{attribute 'linkalways'} 
{attribute 'no_explicit_call' := 'This FB is a CLASS and must be accessed using methods or properties'}
{attribute 'enable_dynamic_creation'}
FUNCTION_BLOCK Node_F_VN_GetAt_UDINT EXTENDS VisionNode
VAR
    ipContainer : _ITcVnContainer;
    nElement : _UDINT(0);
    nIndex : _ULINT(0);
    hrPrev : _HRESULT(S_OK);
    hresult : _HRESULT(S_OK);
END_VAR

METHOD PUBLIC  Clone : I_Node
VAR
	pNode : POINTER TO Node_F_VN_GetAt_UDINT;
END_VAR
pNode := __NEW(Node_F_VN_GetAt_UDINT);
Clone := pNode^;
END_METHOD

METHOD FB_init : BOOL
VAR_INPUT
	bInitRetains : BOOL; // if TRUE, the retain variables are initialized (warm start / cold start)
	bInCopyCode : BOOL;  // if TRUE, the instance afterwards gets moved into the copy code (online change)
END_VAR
AddInput('ipContainer', ipContainer);
AddInput('nIndex', nIndex);
AddInput('hrPrev', hrPrev);
AddOutput('nElement', nElement);
AddOutput('hresult',hresult);
END_METHOD

METHOD PROTECTED OnExecute : HRESULT
hresult.Value := F_VN_GetAt_UDINT(
    ipContainer := ipContainer.Value,
    nElement := nElement.Value,
    nIndex := nIndex.Value,
    hrPrev:= hrPrev.Value);
END_METHOD

METHOD PUBLIC PreExecutionCheck
VAR_INPUT
	Check : I_PreExecutionChecks;
END_VAR
Check.IsTrue(ipContainer.IsValid, 'ipContainer must be a valid container');
Check.IsTrue(ipContainer.HasType(TC_GLOBAL_CONST_LIST.ContainerType_Vector_UDINT), 'ipContainer contains incorrect type');
END_METHOD

END_FUNCTION_BLOCK

(* stored: Version 1.1.0.1, ProductVersion 3.1.4024.13
   POU Node_F_VN_GetAt_UDINT: Id {2d00f5c0-babb-4656-8e87-0f94c86e204e}, SpecialFunc None
   Folder Constructor: Id {6f69d982-705f-4120-94f8-3ecd67ded447}
   Method Clone: Id {933d5c72-0c2b-45e0-b85c-e02e3d1a5cf7}
   Method FB_init: Id {3bb2f294-2d95-47a6-828b-3f1faab18ddc}
   Method OnExecute: Id {056597a0-9a12-4bee-925d-77b0448fbe8e}
   Method PreExecutionCheck: Id {6b2a0c7f-2616-445e-99d8-8f1d63f0bd71} *)
